FUNCTION_BLOCK FB_Turmleuchte
VAR_INPUT
END_VAR
VAR_OUTPUT
END_VAR
VAR
	bA_Summer					AT%Q*:BOOL;
	bA_LampeGruen				AT%Q*:BOOL;
	bA_LampeOrange				AT%Q*:BOOL;
	bA_LampeRot					AT%Q*:BOOL;
	bA_Zaehlen					AT%Q*:BOOL;
	
	tZaehlImpuls:				TP;
	
	bStoerung:					BOOL;
	bWarnung:					BOOL;
	bBetrieb:					BOOL;
	bZaehlen:					BOOL;
	
	bBtnSireneAktivieren:		BOOL;
END_VAR

VAR PERSISTENT
	bSireneAktiviert:			BOOL;
END_VAR

bA_LampeGruen := bBetrieb;
bA_LampeOrange :=bWarnung;
bA_LampeRot := bStoerung;
bA_Summer := bStoerung AND NOT MAIN.bProgStop AND MAIN.bProduzieren AND bSireneAktiviert;

IF			bZaehlen THEN
	tZaehlImpuls.IN := TRUE;
	bZaehlen := FALSE;
ELSE
	tZaehlImpuls.IN := FALSE;
END_IF


tZaehlImpuls(Q => bA_Zaehlen, PT := T#300MS);

IF			bBtnSireneAktivieren THEN
	bBtnSireneAktivieren := FALSE;
	bSireneAktiviert := NOT bSireneAktiviert;
END_IF

METHOD betrieb
VAR_INPUT
END_VAR
bBetrieb := true;
END_METHOD

METHOD reset : BOOL
VAR_INPUT
END_VAR
bStoerung := FALSE;
bWarnung := FALSE;
bBetrieb := FALSE;
END_METHOD

METHOD stoerung
VAR_INPUT
END_VAR
bStoerung := true;
END_METHOD

METHOD warnung
VAR_INPUT
END_VAR
bWarnung := true;
END_METHOD

METHOD zaehlen
VAR_INPUT
END_VAR
bZaehlen := true;
END_METHOD

END_FUNCTION_BLOCK

(* stored: Version 1.1.0.1, ProductVersion 3.1.4024.12
   POU FB_Turmleuchte: Id {cece7395-b725-4bb8-b12d-4ef337d617f5}, SpecialFunc None
   Method betrieb: Id {da15ecb8-6a6f-4a58-bf8c-8bf03339426e}
   Method reset: Id {cbcd39fa-2a22-4a83-b04c-b00c1546002c}
   Method stoerung: Id {027dff04-cd20-420d-be2e-1235c87d31e5}
   Method warnung: Id {cad17de3-6cb2-41a6-a7d7-9cedd702839a}
   Method zaehlen: Id {bb5f0c60-6042-42ae-b185-bf4965766e4b} *)
